// TwinCAT 3 PLC project PLC1
// ProgramVersion: 3.1.4024.12
// libraries:
//   Tc2_Standard, * (Beckhoff Automation GmbH)
//   Tc2_System, * (Beckhoff Automation GmbH)
//   Tc3_Module, * (Beckhoff Automation GmbH)
// project tree:
//   / Class Diagram.TcCD (not stored), Param.TcGVL, PlcTask.TcTTO
//   FBs/ Notification.TcPOU, NotificationCollection.TcPOU, NotificationIterator.TcPOU
//   FUNs/ F_VerboseLogger.TcPOU
//   ITFs/ Collection.TcIO, Iterator.TcIO, Object.TcIO
//   POUs/ MAIN.TcPOU
// real-time tasks:
//   TASK PlcTask: cycle T#10ms, priority 20, ADS port 350

CONFIGURATION PLC1
    RESOURCE PLC ON TwinCAT3
        TASK PlcTask(INTERVAL := T#10ms, PRIORITY := 20);
        PROGRAM MAIN WITH PlcTask : MAIN;
    END_RESOURCE
END_CONFIGURATION

// ---- Param.TcGVL
{attribute 'qualified_only'}
VAR_GLOBAL CONSTANT
	MAX_ITERABLE_ITEMS : INT := 20;
END_VAR

// ---- ITFs/Collection.TcIO
INTERFACE Collection

METHOD createIterator : Iterator
VAR_INPUT
END_VAR
END_METHOD

END_INTERFACE

// ---- ITFs/Iterator.TcIO
INTERFACE Iterator

METHOD current : Object
VAR_INPUT
END_VAR
END_METHOD

METHOD hasNext : BOOL
VAR_INPUT
END_VAR
END_METHOD

METHOD next : Object
VAR_INPUT
END_VAR
END_METHOD

PROPERTY Position : INT
GET
END_GET
END_PROPERTY

METHOD reset : BOOL
VAR_INPUT
END_VAR
END_METHOD

END_INTERFACE

// ---- ITFs/Object.TcIO
INTERFACE Object

METHOD getNotification : STRING
VAR_INPUT
END_VAR
END_METHOD

END_INTERFACE

// ---- POUs/MAIN.TcPOU
PROGRAM MAIN
VAR
    Notifications 	: NotificationCollection;
	n				: Object;
	iterator	  	: Iterator;

	bInit			: BOOL;
	bReset			: BOOL;
	bExecute : BOOL;
	nPosition : INT;
	stext : STRING;
END_VAR

IF NOT bInit THEN
	bInit := TRUE;
	
	Notifications.addItem(str := 'The');
	Notifications.addItem(str := 'quick');
	Notifications.addItem(str := 'brown');
	Notifications.addItem(str := 'fox');
	Notifications.addItem(str := 'jumps');
	Notifications.addItem(str := 'over');
	Notifications.addItem(str := 'the');
	Notifications.addItem(str := 'lazy');
	Notifications.addItem(str := 'dog');
	
	iterator := notifications.createIterator();	
	n := Iterator.current();
	
	nPosition := Iterator.Position;
	stext := CONCAT(TO_STRING(nPosition),n.getNotification()); 

	F_VerboseLogger(stext);
	//	F_VerboseLogger(n.getNotification());
END_IF


IF bExecute THEN
	WHILE(Iterator.hasNext()) DO
		n := Iterator.next();

		nPosition := Iterator.Position;
		stext := CONCAT(TO_STRING(nPosition),n.getNotification()); 
		
		F_VerboseLogger(stext);
	//	F_VerboseLogger(n.getNotification());

	END_WHILE
END_IF
bExecute := FALSE;

IF bReset THEN
	iterator.reset();
	n := Iterator.current();
	
	nPosition := Iterator.Position;
	stext := CONCAT(TO_STRING(nPosition),n.getNotification());
 
	F_VerboseLogger(stext);
	//	F_VerboseLogger(n.getNotification());
	bReset := FALSE;
END_IF

END_PROGRAM

// ---- FBs/NotificationCollection.TcPOU
FUNCTION_BLOCK NotificationCollection IMPLEMENTS Collection
VAR
	numberOfItems 			: INT := 0;
	pNotificationList 		: ARRAY[0..Param.MAX_ITERABLE_ITEMS] OF POINTER TO Notification;
	pNotificationIterator 	: POINTER TO NotificationIterator;
END_VAR

METHOD addItem
VAR_INPUT
	str : STRING;
END_VAR
IF (THIS^.numberOfItems >= Param.MAX_ITERABLE_ITEMS) THEN
	ADSLOGSTR( msgCtrlMask := ADSLOG_MSGTYPE_ERROR, msgFmtStr := 'PLC Msg. : %s', strArg := 'System Full');
ELSE
	THIS^.pNotificationList[THIS^.numberOfItems] := __NEW(Notification(sNotification := str));
	THIS^.numberOfItems := THIS^.numberOfItems + 1;
END_IF
END_METHOD

METHOD createIterator : Iterator
THIS^.pNotificationIterator := __NEW(NotificationIterator(pNotificationList := THIS^.pNotificationList));
createIterator := THIS^.pNotificationIterator^;
END_METHOD

METHOD FB_exit : BOOL
VAR_INPUT
	bInCopyCode : BOOL; // if TRUE, the exit method is called for exiting an instance that is copied afterwards (online change).
END_VAR

VAR
	i: INT;
END_VAR
FOR i:=0 TO Param.MAX_ITERABLE_ITEMS DO
	IF THIS^.pNotificationList[i] <> 0 THEN
		__DELETE(THIS^.pNotificationList[i]);
	END_IF
END_FOR

IF THIS^.pNotificationIterator <> 0 THEN
	__DELETE(THIS^.pNotificationIterator);
END_IF
END_METHOD

METHOD FB_init : BOOL
VAR_INPUT
	bInitRetains : BOOL; // if TRUE, the retain variables are initialized (warm start / cold start)
	bInCopyCode : BOOL;  // if TRUE, the instance afterwards gets moved into the copy code (online change)
END_VAR
END_METHOD

END_FUNCTION_BLOCK

// ---- FBs/Notification.TcPOU
{attribute 'enable_dynamic_creation'}
FUNCTION_BLOCK Notification IMPLEMENTS Object
VAR
	sNotification : STRING;
END_VAR

METHOD FB_init : BOOL
VAR_INPUT
	bInitRetains : BOOL; // if TRUE, the retain variables are initialized (warm start / cold start)
	bInCopyCode : BOOL;  // if TRUE, the instance afterwards gets moved into the copy code (online change)
	sNotification : STRING;
END_VAR
THIS^.sNotification := sNotification;
END_METHOD

METHOD getNotification : STRING
VAR_INPUT
END_VAR
getNotification := THIS^.sNotification;
END_METHOD

END_FUNCTION_BLOCK

// ---- FBs/NotificationIterator.TcPOU
{attribute 'enable_dynamic_creation'}
FUNCTION_BLOCK NotificationIterator IMPLEMENTS Iterator
VAR
	pNotificationList 	: ARRAY[0..Param.MAX_ITERABLE_ITEMS] OF POINTER TO Notification;
	//pNotification 		: POINTER TO Notification; 
	nPosition 			: INT := 0;
END_VAR

METHOD current : Object
VAR
	pNotification 		: POINTER TO Notification; 
END_VAR
pNotification := THIS^.pNotificationList[nPosition];
current := pNotification^;
END_METHOD

METHOD FB_init : BOOL
VAR_INPUT
	bInitRetains : BOOL; // if TRUE, the retain variables are initialized (warm start / cold start)
	bInCopyCode : BOOL;  // if TRUE, the instance afterwards gets moved into the copy code (online change)
	pNotificationList : ARRAY[0..Param.MAX_ITERABLE_ITEMS] OF POINTER TO Notification;
END_VAR
This^.pNotificationList := pNotificationList;
END_METHOD

METHOD hasNext : BOOL
IF (THIS^.pNotificationList[nPosition + 1] <> 16#0000) THEN
	hasNext := TRUE;
ELSE
	hasNext := FALSE;	
END_IF
END_METHOD

METHOD next : Object
VAR
	pNotification 		: POINTER TO Notification; 
END_VAR
THIS^.nPosition := THIS^.nPosition + 1;

pNotification := THIS^.pNotificationList[nPosition];
next := pNotification^;
END_METHOD

PROPERTY Position : INT
GET
Position := nPosition;
END_GET
END_PROPERTY

METHOD reset : BOOL
reset := FALSE;

THIS^.nPosition := 0;
reset := TRUE;
END_METHOD

END_FUNCTION_BLOCK

// ---- FUNs/F_VerboseLogger.TcPOU
FUNCTION F_VerboseLogger : BOOL
VAR_INPUT
	Message : STRING;
END_VAR

ADSLOGSTR( msgCtrlMask := ADSLOG_MSGTYPE_LOG, msgFmtStr := 'Verbose Msg. : %s', strArg := Message);

END_FUNCTION
